Yaskawa INFORM job: R1_W73(0,-90)KM-OK.JBI

/JOB
//NAME R1_W73(0,-90)KM-OK
///FOLDERNAME KRIS-SCIANA
//POS
///NPOS 125,125,0,5,0,0
///TOOL 0
///POSTYPE PULSE
///PULSE
C00000=11593,-146415,-127873,62581,-5873,26851
C00001=11593,-146415,-127873,62581,-5873,26851
C00002=15860,-49558,-83418,34556,78723,17538
C00003=39364,-26345,-85575,16519,90185,-5291
C00004=147283,-72393,-113312,16926,96607,-5809
C00005=195134,-28127,-101278,-17588,107021,-16325
C00006=196593,-28510,-98040,-17951,105146,-15671
C00007=199193,-28868,-96291,-18857,104354,-14874
C00008=199193,-30188,-96097,-18781,103597,-14753
C00009=197154,-28543,-96694,-18094,104427,-15415
C00010=192746,-43760,-104624,-6241,99057,-16360
C00011=193007,-42990,-104186,-6349,99195,-16301
C00012=192363,-44326,-105352,-6087,99193,-16464
C00013=200925,-14879,-84438,-29525,107028,-14613
C00014=200293,-14139,-83890,-29292,106909,-14763
C00015=201919,-15830,-85303,-29907,107314,-14403
C00016=201570,-15502,-86434,-29934,107982,-14688
C00017=200671,-14440,-89150,-30022,109698,-15421
C00018=192950,2156,-79454,-18577,118633,-20488
C00019=192950,286,-79339,-18380,117650,-20314
C00020=194927,-4912,-83051,-20881,114394,-20142
C00021=196902,-8354,-85892,-21560,114705,-19683
C00022=196330,-9532,-85125,-21164,113601,-19618
C00023=195869,-8854,-84676,-21018,113592,-19740
C00024=196774,-8526,-85666,-21473,114474,-19672
C00025=187807,-7281,-86481,-18520,114136,-21933
C00026=187937,-10533,-85938,-18259,112247,-21583
C00027=187937,-11865,-85798,-18150,111512,-21463
C00028=187937,-10533,-85938,-18259,112247,-21583
C00029=186530,-12455,-88007,-17804,112314,-21959
C00030=186400,-15069,-88236,-17592,111145,-21808
C00031=186923,-13891,-87365,-17785,111289,-21695
C00032=186527,-13951,-89739,-17847,112597,-22005
C00033=201570,-15502,-86434,-29934,107982,-14688
C00034=179001,-33440,-106016,-4666,78462,73853
///LIMIT ON
C00035=3105,-143356,-132452,2877,3199,57769
///LIMIT OFF
C00036=-86587,-150737,-134459,-6798,28729,62250
C00037=-131399,-7214,-72083,3711,83263,40842
C00038=-146269,67303,-9377,5564,90450,33302
C00039=-145631,68797,-1102,5257,86110,33285
C00040=-141026,101995,32738,-5649,99342,39108
C00041=-141026,101341,32786,-5643,98977,39126
C00042=-141026,101995,32738,-5649,99342,39108
C00043=-145631,68797,-1102,5257,86110,33285
C00044=-140555,71701,2046,-6219,89775,35418
C00045=-140849,71916,2310,-6090,89706,35342
C00046=-140555,71492,2091,-6219,89641,35426
C00047=-140331,76694,6276,-6317,89753,35483
C00048=-149539,58265,-11906,11869,85930,31880
C00049=-151305,58847,-8753,12757,84538,31255
C00050=-151202,59476,-8019,12708,84398,31270
C00051=-150884,57656,-9820,12551,84528,31372
C00052=-149539,58265,-11906,11869,85930,31880
C00053=-149262,66399,-3614,11741,84994,31868
C00054=-150889,83836,16417,17243,89164,36630
C00055=-144050,68554,2779,-3108,80084,48927
C00056=-141059,77386,10726,-15349,86144,59503
C00057=-138723,76982,8929,-21151,85123,58785
C00058=-137702,72396,-14071,2329,110996,83006
C00059=-149865,70539,-3166,37302,106815,90295
C00060=-149556,126995,74917,40508,122869,64677
C00061=-148868,124992,72077,38926,124371,67238
C00062=-149598,94041,28657,40580,119035,87149
C00063=-150795,83050,15891,42429,112581,85181
C00064=-149711,93084,27395,40793,118526,87011
C00065=-151136,83697,15742,42638,113034,85248
C00066=-150594,72909,2231,38573,107616,90679
C00067=-150213,71758,1658,38407,107286,90692
C00068=-149828,74407,5105,38133,106549,90555
C00069=-149828,77924,4546,38619,108255,85549
C00070=-149753,108545,41516,37203,102627,89159
C00071=-137004,94985,16806,11166,102128,86110
C00072=-124950,77685,-1003,-13641,95870,82133
C00073=-134963,46466,-36080,5562,96270,84421
C00074=-128120,91656,9706,-19888,122036,90872
C00075=-123375,97089,28068,-29445,121182,86580
C00076=-124436,97206,28272,-29371,120812,86275
C00077=-124164,102863,28747,-31764,122767,85309
C00078=-129251,45507,-42900,-7509,106499,54073
C00079=-131399,-7214,-72083,3711,83263,40842
C00080=-86587,-150737,-134459,-6798,28729,62250
C00081=26303,-151670,-134708,7277,28428,55443
C00082=150609,-127208,-136061,10329,34945,54133
C00083=179003,-58532,-100821,-5130,62428,74507
C00084=179976,-59689,-97975,-5966,60150,74939
C00085=179046,-62651,-97471,-5371,58266,74717
C00086=180221,-59219,-97676,-6143,60222,75017
C00087=181399,-62291,-97947,-7114,58903,75497
C00088=182691,-54924,-94207,-7960,60485,75827
C00089=181848,-55913,-95607,-7314,60766,75528
C00090=193229,-20630,-80633,-28206,85002,77205
C00091=193208,-20364,-80778,-28189,85197,77151
C00092=191630,-25188,-83723,-27389,84199,76926
C00093=191427,-27331,-83527,-27331,83060,77134
C00094=191576,-24600,-84066,-27344,84642,76806
C00095=192668,-27231,-84449,-27950,83929,77298
C00096=190232,-31047,-85818,-26733,82301,76949
C00097=190243,-28417,-86415,-26663,83848,76601
C00098=190417,-23791,-87237,-26683,86479,76052
C00099=159326,-66710,-123402,51396,91267,73770
C00100=159322,-93073,-116294,52092,79832,67349
C00101=162473,-91145,-112272,51098,77259,67443
C00102=163034,-88602,-109411,50957,76680,67398
C00103=163692,-89357,-111527,50551,76931,67861
C00104=162236,-92530,-111352,51397,76562,66931
C00105=164396,-94475,-111898,50699,75007,67141
C00106=163105,-90673,-111435,50895,76759,67476
C00107=164703,-89479,-109143,38553,60446,66179
C00108=165663,-89603,-108114,38232,59495,66229
C00109=165421,-87924,-109222,37845,60825,66652
C00110=164006,-90997,-109029,39254,60069,65704
C00111=165166,-88297,-107659,38387,60010,66210
C00112=164224,-89725,-109986,38698,60953,66169
C00113=161176,-91872,-114096,39975,63349,65795
C00114=161178,-67775,-121908,36333,77068,70876
C00115=166243,-48574,-98857,57601,111877,72113
C00116=166229,-47992,-97415,58281,112960,71945
C00117=166127,-50084,-97716,57949,112525,71546
C00118=170915,-50285,-96969,57523,110262,78499
C00119=170916,-50289,-96971,57522,110261,78499
C00120=177188,-46452,-95545,56001,107786,80003
C00121=172595,-49170,-96859,59685,106728,78484
C00122=171487,-80798,-112185,85165,102508,76107
C00123=108277,-148876,-125625,84404,103957,76066
C00124=36161,-141817,-123727,85103,102738,77332
BC00000=148190,850079,1068952
BC00001=148190,1111863,1068952
BC00002=140692,1189228,1068467
BC00003=82735,1188983,1068204
BC00004=379332,1189015,1068204
BC00005=394257,1099256,1068222
BC00006=394257,1095542,1068222
BC00007=394257,1094057,1068222
BC00008=394257,1094057,1068222
BC00009=394257,1094057,1068222
BC00010=394257,1082321,1068222
BC00011=394257,1082321,1068222
BC00012=394257,1082321,1068222
BC00013=394257,1102952,1068222
BC00014=394257,1102952,1068222
BC00015=394257,1102952,1068222
BC00016=394257,1104787,1068222
BC00017=394257,1109374,1068222
BC00018=394257,1109374,1068222
BC00019=394257,1109374,1068222
BC00020=394257,1109374,1068222
BC00021=394257,1109374,1068222
BC00022=394257,1109374,1068222
BC00023=394257,1109374,1068222
BC00024=394257,1109374,1068222
BC00025=394257,1109374,1068222
BC00026=394257,1109374,1068222
BC00027=394257,1109374,1068222
BC00028=394257,1109374,1068222
BC00029=394257,1109374,1068222
BC00030=394257,1109374,1068222
BC00031=394257,1109374,1068222
BC00032=394257,1109374,1068222
BC00033=394257,1104787,1068222
BC00034=394257,1130948,1068222
BC00035=125370,1176627,1068222
BC00036=125370,756629,1068222
BC00037=247706,673691,1068222
BC00038=295256,674297,1068222
BC00039=295256,674297,1068222
BC00040=295256,674297,1068222
BC00041=295256,674297,1068222
BC00042=295256,674297,1068222
BC00043=295256,674297,1068222
BC00044=295256,674297,1068222
BC00045=295256,674297,1068222
BC00046=295256,674297,1068222
BC00047=295256,674297,1068222
BC00048=295256,674297,1068222
BC00049=295256,674297,1068222
BC00050=295256,674297,1068222
BC00051=295256,674297,1068222
BC00052=295256,674297,1068222
BC00053=295256,674297,1068222
BC00054=295256,674297,1068222
BC00055=295256,674297,1068222
BC00056=295256,674296,1068220
BC00057=295256,674297,1068222
BC00058=232213,704134,1068222
BC00059=232213,704134,1068222
BC00060=232213,711089,1068222
BC00061=232213,711089,1068222
BC00062=232213,711089,1068222
BC00063=232213,711089,1068222
BC00064=232213,711089,1068222
BC00065=232213,711089,1068222
BC00066=232213,711089,1068222
BC00067=232213,711089,1068222
BC00068=232213,711089,1068222
BC00069=232213,711089,1068222
BC00070=232213,711089,1068222
BC00071=232213,711089,1068222
BC00072=232213,711089,1068222
BC00073=232213,711089,1068222
BC00074=232213,711089,1068222
BC00075=232213,711089,1068222
BC00076=232213,711089,1068222
BC00077=232213,711089,1068222
BC00078=242849,685414,1068222
BC00079=247706,673691,1068222
BC00080=125370,756629,1068222
BC00081=129018,1145543,1068222
BC00082=393958,1130504,1068220
BC00083=394257,1130962,1068222
BC00084=394257,1126599,1068222
BC00085=394257,1124854,1068222
BC00086=394257,1124854,1068222
BC00087=394257,1124854,1068222
BC00088=394257,1124815,1068222
BC00089=394257,1125687,1068222
BC00090=394257,1130590,1068222
BC00091=394257,1131134,1068222
BC00092=394257,1131179,1068222
BC00093=394257,1130090,1068222
BC00094=394257,1130090,1068222
BC00095=394257,1130090,1068222
BC00096=394257,1130129,1068222
BC00097=394257,1131867,1068222
BC00098=394257,1136206,1068222
BC00099=394257,1054493,1068222
BC00100=394257,1054506,1068222
BC00101=394257,1055792,1068222
BC00102=394257,1056306,1068222
BC00103=394257,1056306,1068222
BC00104=394257,1056306,1068222
BC00105=394257,1056306,1068222
BC00106=394257,1059121,1068222
BC00107=394257,1086901,1068222
BC00108=394257,1086890,1068222
BC00109=394257,1086890,1068222
BC00110=394257,1086890,1068222
BC00111=394257,1083866,1068222
BC00112=394257,1084371,1068222
BC00113=394257,1085752,1068222
BC00114=394257,1085738,1068222
BC00115=394257,1020271,1068222
BC00116=394257,1017944,1068222
BC00117=394257,1017944,1068222
BC00118=394257,1017944,1068222
BC00119=394257,1017944,1068222
BC00120=394257,1017944,1068220
BC00121=394257,1017944,1068218
BC00122=394257,1109426,1068220
BC00123=394257,1109426,1068220
BC00124=229988,732202,1068220
///POSTYPE BASE
///RECTAN
///RCONF 0,0,0,0,0,0,0,0,0,0,0,0,0,0,0,0,0,0,0,0,0,0,0,0
P00006=0.222,-3.123,-1.508,0.0000,0.0000,0.0000
P00023=0.143,-0.036,0.682,0.0000,0.0000,0.0000
P00024=0.145,-0.552,1.326,0.0000,0.0000,0.0000
P00025=-2.003,0.006,0.728,0.0000,0.0000,0.0000
P00026=0.562,-0.002,-0.337,0.0000,0.0000,0.0000
//INST
///DATE 2024/07/24 12:31
///ATTR SC,RW
///GROUP1 RB1,BS1
NOP
'r1_W73(0,-90)
SFTOF
MOVJ C00000 BC00000 VJ=100.00
MOVJ C00001 BC00001 VJ=100.00
MOVJ C00002 BC00002 VJ=100.00
MOVL C00003 BC00003 V=833.3
MOVL C00004 BC00004 V=833.3
MOVL C00005 BC00005 V=500.0
MOVL C00006 BC00006 V=250.0
MOVL C00007 BC00007 V=133.3
REFP 3 C00008 BC00008
CALL JOB:SEARCH-R1
SET P023 P006
SFTON P023
MOVL C00009 BC00009 V=60.0
MOVL C00010 BC00010 V=60.0
REFP 3 C00011 BC00011
CALL JOB:SEARCH-R1
SET P023 P006
SFTON P023
MOVL C00012 BC00012 V=60.0
MOVL C00013 BC00013 V=60.0
REFP 3 C00014 BC00014
CALL JOB:SEARCH-R1
SET P023 P006
SFTON P023
MOVL C00015 BC00015 V=60.0
MOVL C00016 BC00016 V=166.7
MOVL C00017 BC00017 V=166.7
'Path W514
SFTOF
MOVL C00018 BC00018 V=60.0
REFP 3 C00019 BC00019
CALL JOB:SEARCH-R1
SET P025 P006
SFTON P025
MOVL C00020 BC00020 V=60.0
MOVL C00021 BC00021 V=60.0
MOVL C00022 BC00022 V=60.0
REFP 3 C00023 BC00023
CALL JOB:SEARCH-R1
SET P025 P006
SFTOF
MOVL C00024 BC00024 V=60.0
MOVL C00025 BC00025 V=166.7
MOVL C00026 BC00026 V=60.0
REFP 3 C00027 BC00027
CALL JOB:SEARCH-R1
SET P026 P006
SFTON P026
MOVL C00028 BC00028 V=60.0
MOVL C00029 BC00029 V=60.0
MOVL C00030 BC00030 V=60.0
REFP 3 C00031 BC00031
CALL JOB:SEARCH-R1
SET P026 P006
SFTOF
MOVL C00032 BC00032 V=60.0
MOVL C00033 BC00033 V=166.7
SFTON P023
MOVJ C00034 BC00034 VJ=100.00
'POMIAR 2 STRONA
'Path S1141
SFTOF
MOVJ C00035 BC00035 VJ=100.00
MOVJ C00036 BC00036 VJ=100.00
MOVJ C00037 BC00037 VJ=100.00
MOVJ C00038 BC00038 VJ=100.00
MOVL C00039 BC00039 V=100.0
MOVL C00040 BC00040 V=60.0
REFP 3 C00041 BC00041
CALL JOB:SEARCH-R1
SET P024 P006
SFTON P024
MOVL C00042 BC00042 V=60.0
MOVL C00043 BC00043 V=100.0
MOVL C00044 BC00044 V=60.0
REFP 3 C00045 BC00045
CALL JOB:SEARCH-R1
SET P024 P006
SFTON P024
MOVL C00046 BC00046 V=60.0
MOVL C00047 BC00047 V=100.0
MOVL C00048 BC00048 V=100.0
MOVL C00049 BC00049 V=60.0
REFP 3 C00050 BC00050
CALL JOB:SEARCH-R1
SET P024 P006
SFTON P024
MOVL C00051 BC00051 V=60.0
MOVL C00052 BC00052 V=166.7
MOVL C00053 BC00053 V=250.0
SFTOF
SFTOF
SFTON P024
MOVL C00054 BC00054 V=166.7 PL=0
MACRO1 MJ#(0) ARGF12
ARCON
MOVL C00055 BC00055 V=9.2
MOVL C00056 BC00056 V=9.2
ARCOF
MOVL C00057 BC00057 V=100.0
MOVL C00058 BC00058 V=250.0
MOVJ C00059 BC00059 VJ=100.00
'COMMENT
'COMMENT
SFTOF
SFTON P024
MOVL C00060 BC00060 V=250.0
MOVL C00061 BC00061 V=166.7 PL=0
MACRO1 MJ#(0) ARGF12
ARCON
MOVL C00062 BC00062 V=8.3
ARCOF
MOVL C00063 BC00063 V=133.3
ARCON
MOVL C00064 BC00064 V=9.2
ARCOF
MOVL C00065 BC00065 V=166.7
MOVL C00066 BC00066 V=166.7
'COMMENT
'COMMENT
SFTOF
SFTON P024
MOVL C00067 BC00067 V=100.0 PL=0
MACRO1 MJ#(0) ARGF12
ARCON
MOVL C00068 BC00068 V=9.2
ARCOF
SFTOF
MOVL C00069 BC00069 V=250.0
MOVJ C00070 BC00070 VJ=100.00
MOVJ C00071 BC00071 VJ=100.00
MOVJ C00072 BC00072 VJ=100.00
MOVJ C00073 BC00073 VJ=100.00
MOVJ C00074 BC00074 VJ=100.00
'COMMENT
'COMMENT
SFTOF
SFTON P024
MOVL C00075 BC00075 V=166.7 PL=0
MACRO1 MJ#(0) ARGF12
ARCON
MOVL C00076 BC00076 V=11.7
ARCOF
MOVL C00077 BC00077 V=166.7
SFTOF
MOVJ C00078 BC00078 VJ=100.00
MOVJ C00079 BC00079 VJ=100.00
MOVJ C00080 BC00080 VJ=100.00
MOVJ C00081 BC00081 VJ=100.00
MOVJ C00082 BC00082 VJ=100.00
'KONIEC POMIAR 2 STRONA
MOVL C00083 BC00083 V=500.0
MOVL C00084 BC00084 V=166.7
SFTON P023
MOVL C00085 BC00085 V=100.0 PL=0
REFP 1 C00086 BC00086
REFP 2 C00087 BC00087
MACRO1 MJ#(0) ARGF12
ARCON
MOVL C00088 BC00088 V=9.2
ARCOF
MOVL C00089 BC00089 V=166.7
SFTOF
MOVL C00090 BC00090 V=250.0
MOVL C00091 BC00091 V=250.0
SFTON P026
MOVL C00092 BC00092 V=250.0
MOVL C00093 BC00093 V=166.7 PL=0
REFP 1 C00094 BC00094
REFP 2 C00095 BC00095
MACRO1 MJ#(0) ARGF12
ARCON
MOVL C00096 BC00096 V=9.2
ARCOF
MOVL C00097 BC00097 V=250.0
MOVL C00098 BC00098 V=333.3
SFTOF
'Path W513
SFTOF
SFTON P023
MOVJ C00099 BC00099 VJ=100.00
MOVL C00100 BC00100 V=333.3
MOVL C00101 BC00101 V=333.3
MOVL C00102 BC00102 V=166.7 PL=0
REFP 1 C00103 BC00103
REFP 2 C00104 BC00104
MACRO1 MJ#(0) ARGF12
ARCON
MOVL C00105 BC00105 V=9.5
ARCOF
MOVL C00106 BC00106 V=166.7
MOVL C00107 BC00107 V=250.0
MOVL C00108 BC00108 V=100.0 PL=0
REFP 1 C00109 BC00109
REFP 2 C00110 BC00110
MACRO1 MJ#(0) ARGF12
ARCON
MOVL C00111 BC00111 V=9.5
ARCOF
MOVL C00112 BC00112 V=166.7
MOVL C00113 BC00113 V=500.0
MOVL C00114 BC00114 V=833.3
SFTOF
MOVJ C00115 BC00115 VJ=100.00
SFTON P026
MACRO1 MJ#(0) ARGF12
MOVJ C00116 BC00116 VJ=100.00
MOVL C00117 BC00117 V=166.7
ARCON
MOVL C00118 BC00118 V=9.2
MOVL C00119 BC00119 V=9.2
SFTON P025
MOVL C00120 BC00120 V=9.2
ARCOF
MOVJ C00121 BC00121 VJ=100.00
SFTOF
MOVJ C00122 BC00122 VJ=100.00
MOVJ C00123 BC00123 VJ=100.00
MOVJ C00124 BC00124 VJ=100.00
END
